INCR:=FALSE;
DECR:=FALSE;
IF IN_A <> IN_A_LAST THEN (*Flanke auf A:*)
	IF IN_A THEN(* Positive Flanke Spur A*)
		IF IN_B THEN DECR:=TRUE;
		ELSE INCR:=TRUE;
		END_IF
	ELSE (*negative Flanke auf A*)
		IF IN_B THEN INCR:=TRUE;
		ELSE DECR:=TRUE;
		END_IF
	END_IF
ELSIF IN_B <> IN_B_LAST THEN (*Flanke auf B:*)
	IF IN_B THEN(* Positive Flanke Spur B*)
		IF IN_A THEN INCR:=TRUE;
		ELSE DECR:=TRUE;
		END_IF
	ELSE (*negative Flanke auf B*)
		IF IN_A THEN DECR:=TRUE;
		ELSE INCR:=TRUE;
		END_IF
	END_IF
END_IF

(*Stillstandsüberwachung*)
IF (VOR_OUT AND NOT INCR) OR (ZUR_OUT AND NOT DECR) THEN (*Überwachung auf Mechanische blockade*)
	T_STILLST:=T_STILLST + T_ZYKL;
ELSE
	T_STILLST:=0;
END_IF

IF (VOR_OUT OR ZUR_OUT ) AND (IN_A=IN_A_LAST) THEN (*Überwachung SPUR A*)
	T_STILLST_A:=T_STILLST_A + T_ZYKL;
ELSE
	T_STILLST_A:=0;
END_IF

IF (VOR_OUT OR ZUR_OUT ) AND (IN_B=IN_B_LAST) THEN (*Überwachung SPUR B*)
	T_STILLST_B:=T_STILLST_B + T_ZYKL;
ELSE
	T_STILLST_B:=0;
END_IF
DAT_TO_PLC.STILL:=(T_STILLST > (2*T_pro_INC)) OR MAX(T_STILLST_A,T_STILLST_B)>(4*T_pro_INC); (*Stillstandsüberwachungszeit abgelaufen: Flanke nicht nach doppelter Zeit gekommen oder Spur A nicht nach doppelter (4*Increment)gekommen->SET Stillstand*)



IF INCR THEN IstIncr:=IstIncr+1;T_seit_Letzt_EncFl:=0.0;
ELSIF DECR THEN IstIncr:=IstIncr-1;T_seit_Letzt_EncFl:=T_pro_INC;
END_IF

(*Zeitberechnung seit letzter Encoderflanke*)
IF VOR_OUT THEN T_seit_Letzt_EncFl:=MIN((T_seit_Letzt_EncFl+T_ZYKL),T_pro_INC);
ELSIF ZUR_OUT THEN T_seit_Letzt_EncFl:=MAX((T_seit_Letzt_EncFl-T_ZYKL),0);
END_IF

(*############# Referenzmodus: ohne Nullspur  #############*)
IF DAT_FROM_PLC.REF THEN
	IF REFSTATUS=0 THEN (*Referenzfahrt hat noch nicht begonnen*)
		SYNC:=FALSE;(*Sync löschen bei Anwahl von Ref-Modus*)
		REFSTATUS:=1;(*Refstatus: suche Endschalter*)
	ELSIF REFSTATUS=1 AND EREF THEN REFSTATUS:=2; (*Wenn Status=suche Endschalter und EREF belegt, dann Status=2*)
	ELSIF REFSTATUS=2 AND NOT EREF THEN REFSTATUS:=3; (*negative Flanke Endschalter: Refstatus=3: suche erste Flanke Encodersignale*)
	ELSIF REFSTATUS=3 AND (INCR OR DECR) THEN REFSTATUS:=7;(*negative Flanke Endschalter: Refstatus=7 (fertig, Istwert neu setzen*)
		IstIncr:=0;
		SYNC:=TRUE;
	END_IF
ELSE REFSTATUS:=0;(*Wenn nicht REF-Modus, dann REFSTATUS=0*)
END_IF

(*Istposition setzen*)
IF DAT_FROM_PLC.SETPOS THEN
	IstIncr:=0;
	T_seit_Letzt_EncFl:=0.0;
	SYNC:=TRUE;
END_IF



(*#################  Ermittlung des Geberistwertes. Die Zeitinterpolierte Strecke wird limitiert auf IBW (Weg zwischen 2 Incrementen, sollte keine Flanke mehr von A oder B einfallen, löst Stillstandsüberwachung aus da der Encoder nicht Zählt ################################## *)
IstPos:=DAT_FROM_PLC.REFPOS+IBW*(IstIncr+T_seit_Letzt_EncFl/T_pro_INC); (*Refposition + IstPosition = GANZE INCREMENTE + Teilincremente (Zeitinterpolation*)


(*############################## Achsen-Steuerung ##############################################################*)
PEH:=FALSE; (*PEH mit FALSE initialisieren*)

(*################################ REFERENZFAHRT ################################################*)
IF DAT_FROM_PLC.REF AND NOT SYNC THEN
	IF REFSTATUS=1 THEN V_SOLL:=REFVEL1;
	ELSE V_SOLL:=REFVEL2;
	END_IF

(*########################## Positionieren auf Sollposition######################################*)
(*POSITIONIEREN POSITIONIEREN POSITIONIEREN POSITIONIEREN POSITIONIEREN POSITIONIEREN POSITIONIEREN POSITIONIEREN *)
ELSIF DAT_FROM_PLC.Start_Pos THEN
	Zieldiff_Pos:=DAT_FROM_PLC.Sollpos-IstPos;(*Reelle momentane Differenz zum Ziel*)
	DAT_TO_PLC.RET_SollPos:=DAT_FROM_PLC.Sollpos;
	IF ABS(Zieldiff_Pos)>S_STOP THEN (*Positionieren, STOP-Fenster noch nicht erreicht*)
		IF Zieldiff_Pos > 0 THEN (*vorwärts positionieren*)
			V_SOLL:=1; (*langsam vor*)
		ELSE (*rückwärts positionieren*)
			V_SOLL:=-1; (*langsam zurück*)
		END_IF
	ELSE (*S_STOP-Fenster bereits erreicht*)
		V_SOLL:=0; (*keine Startfreigabe (Positionierung bereits ausgeführt), also STOP*)
		PEH:=TRUE;
		V_SOLL:=0;
	END_IF

(*################### JOG-Betrieb mit konstanter Geschwindigkeit ohne Startrampe ###################*)
(* JOG JOG JOG JOG JOG JOG JOG JOG JOG JOG JOG JOG JOG JOG JOG JOG JOG JOG JOG JOG JOG JOG JOG JOG JOG JOG JOG *)
ELSIF DAT_FROM_PLC.JOGFW THEN
	V_SOLL:=DAT_FROM_PLC.V_JOG;

ELSIF DAT_FROM_PLC.JOGBW THEN
	V_SOLL:=-DAT_FROM_PLC.V_JOG;

(*####################### Anhalten, keine Bedingung erfüllt##########################################*)
(* HALT HALT HALT HALT HALT HALT HALT HALT HALT HALT HALT HALT HALT HALT HALT HALT HALT HALT HALT HALT HALT HALT *)
ELSE V_SOLL:=0;
END_IF


(*########## Berechnung der Ausgänge ###############*)
IF V_SOLL > 0 THEN (*Sollgeschwindigkeit vor*)
	IF TIME_ZUR=0 THEN (*keine Richtungsumkehr, rückwärts-Wartezeit ist abgelaufen*)
		(*positionieren vor*)
		TIME_VOR:=WAITTIME_INV;(*Wartezeit laden*)
		DAT_TO_PLC.VEL_IST:=1;
	ELSE (*Rückwärts-Wartezeit läuft noch*)
		DAT_TO_PLC.VEL_IST:=0;
	END_IF
ELSIF V_SOLL < 0 THEN(*Sollgeschwindigkeit negativ*)
	IF TIME_VOR=0 THEN (*keine Richtungsumkehr, vorwärts-Wartezeit ist abgelaufen*)
		(*positionieren zurück*)
		TIME_ZUR:=WAITTIME_INV;(*Wartezeit "zurück" laden*)
		DAT_TO_PLC.VEL_IST:=-1;
	ELSE (*vorwärts-Wartezeit läuft noch*)
		DAT_TO_PLC.VEL_IST:=0;
	END_IF
ELSE (*Sollgeschwindigkeit = 0, also STOP*)
	DAT_TO_PLC.VEL_IST:=0;
END_IF
(*Wartezeit decrementieren*)
TIME_VOR:=MAX((TIME_VOR-T_ZYKL),0);TIME_ZUR:=MAX((TIME_ZUR-T_ZYKL),0);
(*Zyklusverz. Var.*)


(*Ausgangsvariablen übergeben*)
DAT_TO_PLC.IstPos:=IstPos;
DAT_TO_PLC.SYNC:=SYNC;
DAT_TO_PLC.PEH:=PEH;
(*Ausgänge setzen*)
VOR_OUT:=DAT_TO_PLC.VEL_IST>0;
ZUR_OUT:=DAT_TO_PLC.VEL_IST<0;

Start_Pos_LAST:=DAT_FROM_PLC.Start_Pos;
IN_A_LAST:=IN_A;
IN_B_LAST:=IN_B;

END_FUNCTION_BLOCK
